PROGRAM ST20_VisionManualControl
VAR
END_VAR

IF G_MachineControl.stMachineOperateMode.MANUAL THEN
	
	IF G_Manual.M20_bVisionTrayFiducial1 THEN
		G_Vision.V20_bRespone := FALSE;
		G_Vision.V20_sSendCmd := 'TRG,0';
		G_Vision.V20_bTrigger := TRUE;
		G_Manual.M20_bVisionTrayFiducial1 := FALSE;	
	END_IF
	
	IF G_Manual.M20_bVisionTrayFiducial2 THEN
		G_Vision.V20_bRespone := FALSE;
		G_Vision.V20_sSendCmd := 'TRG,1';
		G_Vision.V20_bTrigger := TRUE;
		G_Manual.M20_bVisionTrayFiducial2 := FALSE;	
	END_IF
	
	IF G_Manual.M20_bVisionPalletFiducial1 THEN
		G_Vision.V20_bRespone := FALSE;
		G_Vision.V20_sSendCmd := 'TRG,2';
		G_Vision.V20_bTrigger := TRUE;
		G_Manual.M20_bVisionPalletFiducial1 := FALSE;	
	END_IF
	
	IF G_Manual.M20_bVisionPalletFiducial2 THEN
		G_Vision.V20_bRespone := FALSE;
		G_Vision.V20_sSendCmd := 'TRG,3';
		G_Vision.V20_bTrigger := TRUE;
		G_Manual.M20_bVisionPalletFiducial2 := FALSE;	
	END_IF
	
END_IF

END_PROGRAM

(* stored: Version 1.1.0.1, ProductVersion 3.1.4024.11
   POU ST20_VisionManualControl: Id {f3db2985-5627-426a-b1d7-32ec64798b2d}, SpecialFunc None *)
